Staubli VAL3: getDistance.pgx

public program getDistance(tool x_tTool, num& x_nDistance[], bool x_bCycle, num x_nIndex)
  local point l_pPoint
  local num l_nValue
  local trsf l_trsfEmpty
  local point l_pActual
  local point l_pPrev
begin
  // first point
  if x_nIndex==0
    x_nDistance=10
    return
  else
    //
    // get the point
    //
    call getPoint(l_pActual,x_bCycle,x_nIndex)
    call getPoint(l_pPrev,x_bCycle,x_nIndex-1)
    if x_bCycle
      // an other one

      switch pt:tTraj[sItemCycle].tData[x_nIndex].nType
        case 0
          // appro
          x_nDistance=distance(position(l_pPrev,world),position(l_pActual,world))
        break
        case 1
          // point
          x_nDistance=distance(l_pPrev.trsf,l_trsfEmpty)
        break
        case 2
          // depart
          if pt:tTraj[sItemCycle].tData[x_nIndex-1].nType==1
            x_nDistance=distance(l_trsfEmpty,l_pActual.trsf)
          else
            x_nDistance=distance(position(l_pPrev,world),position(l_pActual,world))
          endIf
        break
      endSwitch
    else
      // an other one
      switch pEditPoint[x_nIndex].tData.nType
        case 0
          // appro
          x_nDistance=distance(position(l_pPrev,world),position(l_pActual,world))
        break
        case 1
          // point
          x_nDistance=distance(l_pPrev.trsf,l_trsfEmpty)
        break
        case 2
          // depart
          if pEditPoint[x_nIndex-1].tData.nType==1
            x_nDistance=distance(l_trsfEmpty,l_pActual.trsf)
          else
            x_nDistance=distance(position(l_pPrev,world),position(l_pActual,world))
          endIf
        break
      endSwitch
    endIf
  endIf
end
